// TIA Portal V19 export
TYPE "LEXCHANGETRAY_typePlasticEm5_toHandlingXyzReq"
// stored: Access Published
   STRUCT
      transferEnable : Bool;   // 请求排料排料
   END_STRUCT;
END_TYPE
